(* PLC project project, Beckhoff Automation GmbH TwinCAT PLC Control 3.5.6.1 *)
(* stored: creationDateTime 2016-08-11T14:04:35.7870087, modificationDateTime 2016-08-11T14:04:35.7940091 *)

TYPE IOStruct :
STRUCT
	input_one : BOOL;
	input_two : BOOL;
	input_three : BOOL;
	input_four : BOOL;
	input_five : BOOL;
	input_six : BOOL;
END_STRUCT
END_TYPE

FUNCTION IO_aggregation : BOOL
VAR_INPUT
END_VAR
VAR
END_VAR

                  //Jedem Wert einen sensor zuweißen 
//Byte von 0-7; Position 0 am ende!!!!
//Z.B:

//IO_data.input_v.1 := GVL.in_MagazinNotaus;
//IO_data.input_one := NOT GVL.in_SortierbandNotaus;
//IO_data.input_two := NOT GVL.in_MagazinNotaus;
//IO_data.input_three := NOT GVL.in_StempelNotaus;
//IO_data.input_four := Main.Crane.Crane_SoftwareEmergency;
//IO_data.input_five := Main.Stamp.Stamp_SoftwareEmergency;
//IO_data.input_six := Main.PicAlpha.PicAlpha_SoftwareEmergency;
                
END_FUNCTION

PROGRAM MAIN
VAR		
	XPPU : XPPU;
END_VAR

                  XPPU();


//Für ADS
IO_aggregation();
                
END_PROGRAM

FUNCTION_BLOCK BistableCylinder
VAR_INPUT		
	SFCReset : BOOL;
END_VAR
VAR_OUTPUT
END_VAR
VAR	
	DI_Extended AT %I* : BOOL;
	DI_Retracted AT %I* : BOOL;
	DO_Extend AT %Q* : BOOL;
	DO_Retract AT %Q* : BOOL;
END_VAR

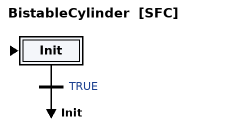
INITIAL_STEP Init:
END_STEP
TRANSITION FROM Init TO Init
  := TRUE;
END_TRANSITION

ACTION ACT_Retract:
                      DO_Extend:=FALSE;
DO_Retract:=TRUE;
                    
END_ACTION

ACTION ACT_Extend:
                      DO_Retract:=FALSE;
DO_Extend:=TRUE;
                    
END_ACTION
END_FUNCTION_BLOCK

FUNCTION_BLOCK MonostableCylinder
VAR_INPUT	
	SFCReset : BOOL;
END_VAR	
VAR_OUTPUT	
END_VAR
VAR	
	DI_Extended AT %I* : BOOL;
	DI_Retracted AT %I* : BOOL;
	
	DO_Extend AT %Q* : BOOL;
END_VAR

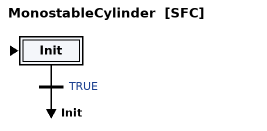
INITIAL_STEP Init:
END_STEP
TRANSITION FROM Init TO Init
  := TRUE;
END_TRANSITION

ACTION ACT_Extend:
                      DO_Extend:=TRUE;
                    
END_ACTION

ACTION ACT_Retract:
                      DO_Extend:=FALSE;
                    
END_ACTION
END_FUNCTION_BLOCK

FUNCTION_BLOCK Motor
VAR_INPUT	
	SFCReset : BOOL;
END_VAR
VAR_OUTPUT	
END_VAR
VAR	
	//Hardware
	DO_Forwards AT %Q* : BOOL;
	DO_Backwards AT %Q* : BOOL;
END_VAR

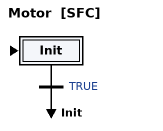
INITIAL_STEP Init:
END_STEP
TRANSITION FROM Init TO Init
  := TRUE;
END_TRANSITION

ACTION ACT_TurnBackwards:
                      DO_Forwards:=FALSE;
DO_Backwards:=TRUE;
                    
END_ACTION

ACTION ACT_Stop:
                      DO_Forwards:=FALSE;
DO_Backwards:=FALSE;
                    
END_ACTION

ACTION ACT_TurnForwards:
                      DO_Backwards:=FALSE;
DO_Forwards:=TRUE;
                    
END_ACTION
END_FUNCTION_BLOCK

FUNCTION_BLOCK Switch
VAR_INPUT	
	SFCReset : BOOL;
END_VAR	
VAR_OUTPUT		
END_VAR
VAR	
	//Hardware
	DI_Extended AT %I* : BOOL;
	DI_Retracted AT %I* : BOOL;	
	DO_Extend AT %Q* : BOOL;
END_VAR

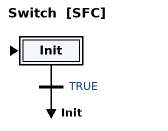
INITIAL_STEP Init:
END_STEP
TRANSITION FROM Init TO Init
  := TRUE;
END_TRANSITION

ACTION ACT_Extend:
                      DO_Extend:=TRUE;
                    
END_ACTION

ACTION ACT_Retract:
                      DO_Extend:=FALSE;
                    
END_ACTION
END_FUNCTION_BLOCK

FUNCTION_BLOCK VacuumGripper
VAR_INPUT	
	SFCReset : BOOL;
END_VAR
VAR_OUTPUT	
END_VAR
VAR	
	//Hardware
	DI_TakenIn AT %I* : BOOL;
	DO_Intake AT %Q* : BOOL;
END_VAR

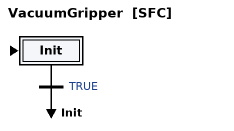
INITIAL_STEP Init:
END_STEP
TRANSITION FROM Init TO Init
  := TRUE;
END_TRANSITION

ACTION ACT_Intake:
                      DO_Intake:=TRUE;
                    
END_ACTION

ACTION ACT_Release:
                      DO_Intake:=FALSE;
                    
END_ACTION
END_FUNCTION_BLOCK

FUNCTION_BLOCK Crane
VAR_INPUT
	LiftingCylinder : MonostableCylinder;
	Gripper : VacuumGripper;			
	//Software
	Crane_SoftwareEmergency : BOOL;
	SFCReset : BOOL;
	InitCompleted : BOOL;
	LSC_AllowedToOperate : BOOL;
	Stamp_AllowedToOperate : BOOL;
	EmergencyHandeled : BOOL;	
END_VAR
VAR_OUTPUT	
	//Software
	Crane_WPPickedUp : BOOL;
	Crane_WPWeight_Light : BOOL;
	Crane_WPWeight_Medium : BOOL;
	Crane_WPWeight_Heavy : BOOL;
	AtStack : BOOL := FALSE;
	AtConveyor : BOOL := FALSE;
	AtStamp : BOOL := FALSE;	
END_VAR
VAR		
	//Hardware	
	Crane_OnStack AT %I* : BOOL;
	Crane_OnConveyor AT %I* : BOOL;
	Crane_OnStamp AT %I* : BOOL;	
	CraneTurnClockwise AT %Q* : BOOL;
	CraneTurnCounterclockwise AT %Q* : BOOL;
	
	//Software
	Timer : TON;	
	AutomaticExecuteAktive : BOOL;
END_VAR

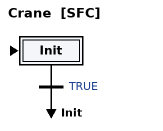
INITIAL_STEP Init:
END_STEP
TRANSITION FROM Init TO Init
  := TRUE;
END_TRANSITION

ACTION ACT_EmergencyStop:
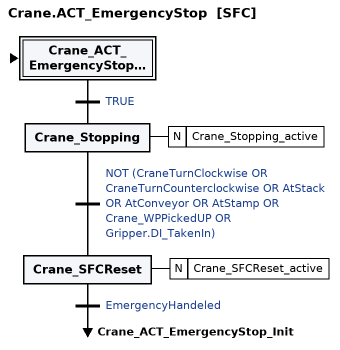
INITIAL_STEP Crane_ACT_EmergencyStop_Init:
END_STEP
TRANSITION FROM Crane_ACT_EmergencyStop_Init TO Crane_Stopping
  := TRUE;
END_TRANSITION
STEP Crane_Stopping:
  Crane_Stopping_active(N);
END_STEP
TRANSITION FROM Crane_Stopping TO Crane_SFCReset
  := NOT (CraneTurnClockwise OR CraneTurnCounterclockwise OR AtStack OR AtConveyor OR AtStamp OR Crane_WPPickedUP OR Gripper.DI_TakenIn);
END_TRANSITION
STEP Crane_SFCReset:
  Crane_SFCReset_active(N);
END_STEP
TRANSITION FROM Crane_SFCReset TO Crane_ACT_EmergencyStop_Init
  := EmergencyHandeled;
END_TRANSITION
END_ACTION

ACTION ACT_AutomaticExecute:
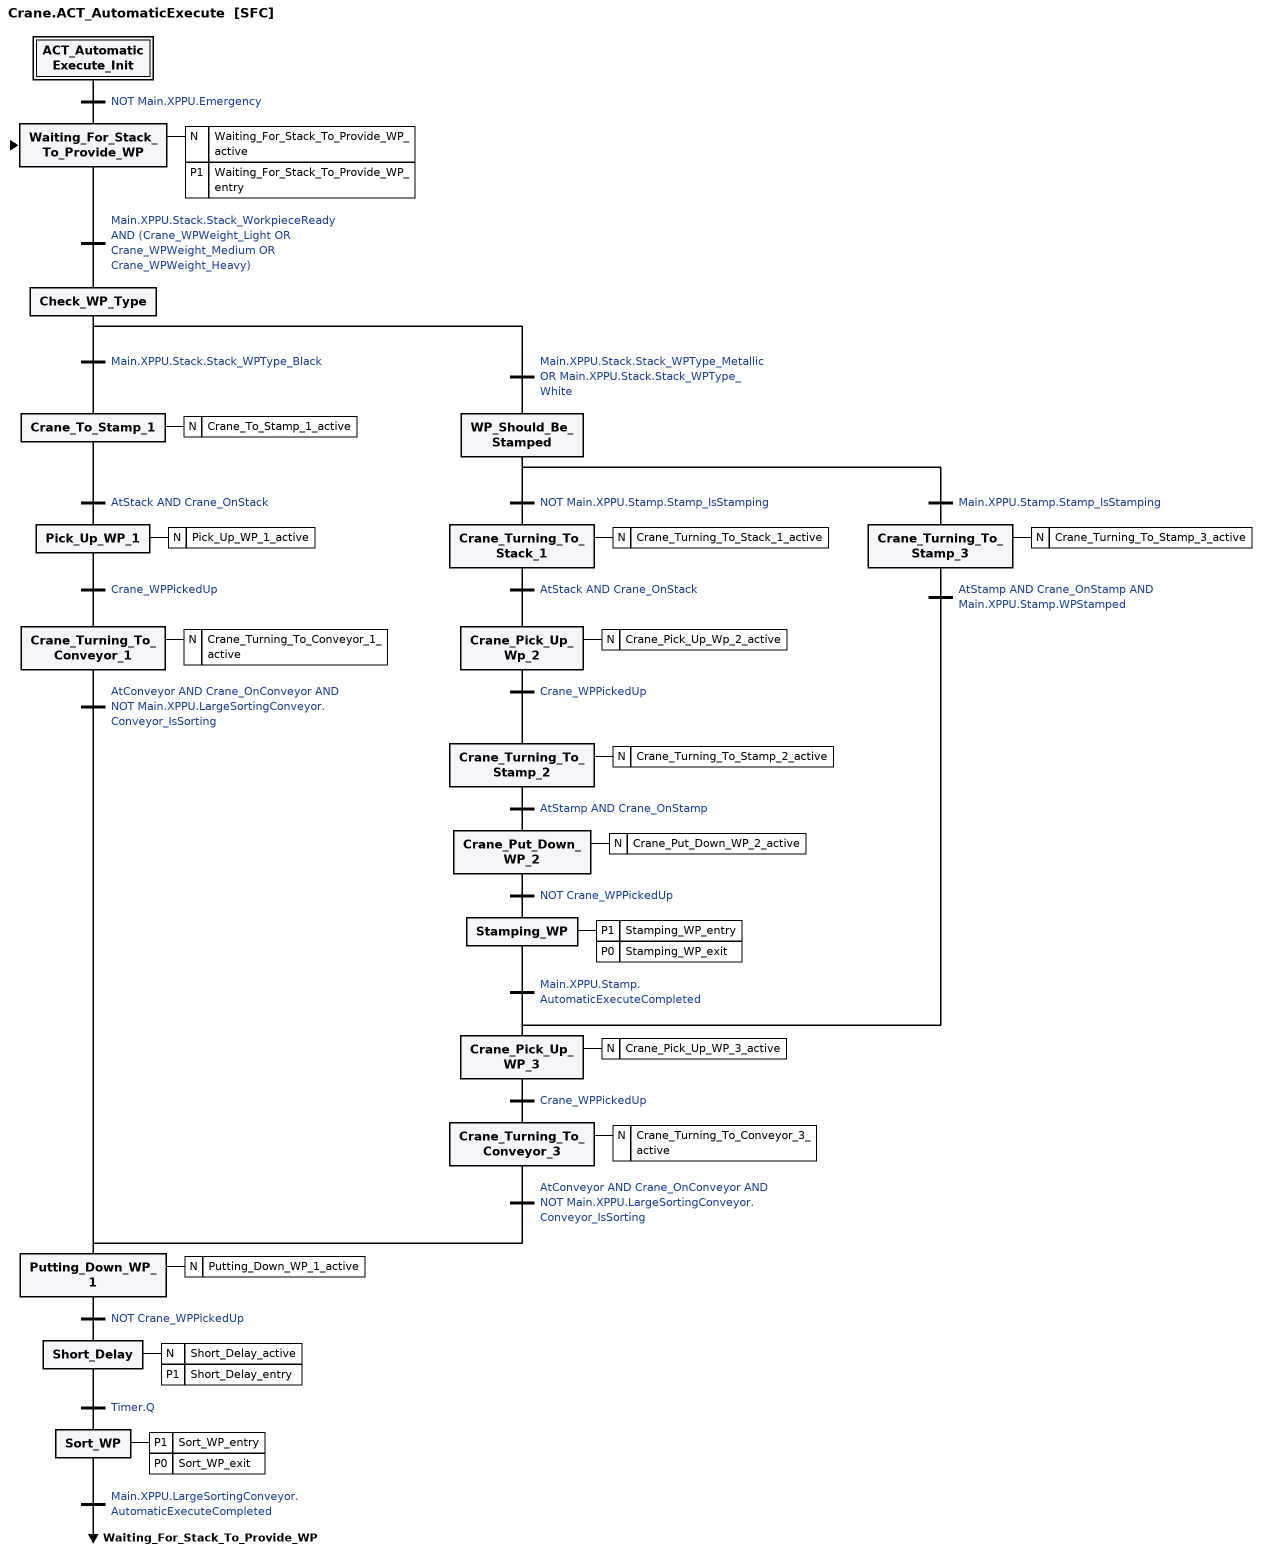
INITIAL_STEP ACT_AutomaticExecute_Init:
END_STEP
TRANSITION FROM ACT_AutomaticExecute_Init TO Waiting_For_Stack_To_Provide_WP
  := NOT Main.XPPU.Emergency;
END_TRANSITION
STEP Waiting_For_Stack_To_Provide_WP:
  Waiting_For_Stack_To_Provide_WP_active(N);
  Waiting_For_Stack_To_Provide_WP_entry(P1);
END_STEP
TRANSITION FROM Waiting_For_Stack_To_Provide_WP TO Check_WP_Type
  := Main.XPPU.Stack.Stack_WorkpieceReady AND (Crane_WPWeight_Light OR Crane_WPWeight_Medium OR Crane_WPWeight_Heavy);
END_TRANSITION
STEP Check_WP_Type:
END_STEP
TRANSITION FROM Check_WP_Type TO Crane_To_Stamp_1
  := Main.XPPU.Stack.Stack_WPType_Black;
END_TRANSITION
TRANSITION FROM Check_WP_Type TO WP_Should_Be_Stamped
  := Main.XPPU.Stack.Stack_WPType_Metallic OR Main.XPPU.Stack.Stack_WPType_White;
END_TRANSITION
STEP Crane_To_Stamp_1:
  Crane_To_Stamp_1_active(N);
END_STEP
TRANSITION FROM Crane_To_Stamp_1 TO Pick_Up_WP_1
  := AtStack AND Crane_OnStack;
END_TRANSITION
STEP Pick_Up_WP_1:
  Pick_Up_WP_1_active(N);
END_STEP
TRANSITION FROM Pick_Up_WP_1 TO Crane_Turning_To_Conveyor_1
  := Crane_WPPickedUp;
END_TRANSITION
STEP Crane_Turning_To_Conveyor_1:
  Crane_Turning_To_Conveyor_1_active(N);
END_STEP
TRANSITION FROM Crane_Turning_To_Conveyor_1 TO Putting_Down_WP_1
  := AtConveyor AND Crane_OnConveyor AND NOT Main.XPPU.LargeSortingConveyor.Conveyor_IsSorting;
END_TRANSITION
STEP Putting_Down_WP_1:
  Putting_Down_WP_1_active(N);
END_STEP
TRANSITION FROM Putting_Down_WP_1 TO Short_Delay
  := NOT Crane_WPPickedUp;
END_TRANSITION
STEP Short_Delay:
  Short_Delay_active(N);
  Short_Delay_entry(P1);
END_STEP
TRANSITION FROM Short_Delay TO Sort_WP
  := Timer.Q;
END_TRANSITION
STEP Sort_WP:
  Sort_WP_entry(P1);
  Sort_WP_exit(P0);
END_STEP
TRANSITION FROM Sort_WP TO Waiting_For_Stack_To_Provide_WP
  := Main.XPPU.LargeSortingConveyor.AutomaticExecuteCompleted;
END_TRANSITION
STEP WP_Should_Be_Stamped:
END_STEP
TRANSITION FROM WP_Should_Be_Stamped TO Crane_Turning_To_Stack_1
  := NOT Main.XPPU.Stamp.Stamp_IsStamping;
END_TRANSITION
TRANSITION FROM WP_Should_Be_Stamped TO Crane_Turning_To_Stamp_3
  := Main.XPPU.Stamp.Stamp_IsStamping;
END_TRANSITION
STEP Crane_Turning_To_Stack_1:
  Crane_Turning_To_Stack_1_active(N);
END_STEP
TRANSITION FROM Crane_Turning_To_Stack_1 TO Crane_Pick_Up_Wp_2
  := AtStack AND Crane_OnStack;
END_TRANSITION
STEP Crane_Pick_Up_Wp_2:
  Crane_Pick_Up_Wp_2_active(N);
END_STEP
TRANSITION FROM Crane_Pick_Up_Wp_2 TO Crane_Turning_To_Stamp_2
  := Crane_WPPickedUp;
END_TRANSITION
STEP Crane_Turning_To_Stamp_2:
  Crane_Turning_To_Stamp_2_active(N);
END_STEP
TRANSITION FROM Crane_Turning_To_Stamp_2 TO Crane_Put_Down_WP_2
  := AtStamp AND Crane_OnStamp;
END_TRANSITION
STEP Crane_Put_Down_WP_2:
  Crane_Put_Down_WP_2_active(N);
END_STEP
TRANSITION FROM Crane_Put_Down_WP_2 TO Stamping_WP
  := NOT Crane_WPPickedUp;
END_TRANSITION
STEP Stamping_WP:
  Stamping_WP_entry(P1);
  Stamping_WP_exit(P0);
END_STEP
TRANSITION FROM Stamping_WP TO Crane_Pick_Up_WP_3
  := Main.XPPU.Stamp.AutomaticExecuteCompleted;
END_TRANSITION
STEP Crane_Turning_To_Stamp_3:
  Crane_Turning_To_Stamp_3_active(N);
END_STEP
TRANSITION FROM Crane_Turning_To_Stamp_3 TO Crane_Pick_Up_WP_3
  := AtStamp AND Crane_OnStamp AND Main.XPPU.Stamp.WPStamped;
END_TRANSITION
STEP Crane_Pick_Up_WP_3:
  Crane_Pick_Up_WP_3_active(N);
END_STEP
TRANSITION FROM Crane_Pick_Up_WP_3 TO Crane_Turning_To_Conveyor_3
  := Crane_WPPickedUp;
END_TRANSITION
STEP Crane_Turning_To_Conveyor_3:
  Crane_Turning_To_Conveyor_3_active(N);
END_STEP
TRANSITION FROM Crane_Turning_To_Conveyor_3 TO Putting_Down_WP_1
  := AtConveyor AND Crane_OnConveyor AND NOT Main.XPPU.LargeSortingConveyor.Conveyor_IsSorting;
END_TRANSITION
END_ACTION

ACTION ACT_Init:
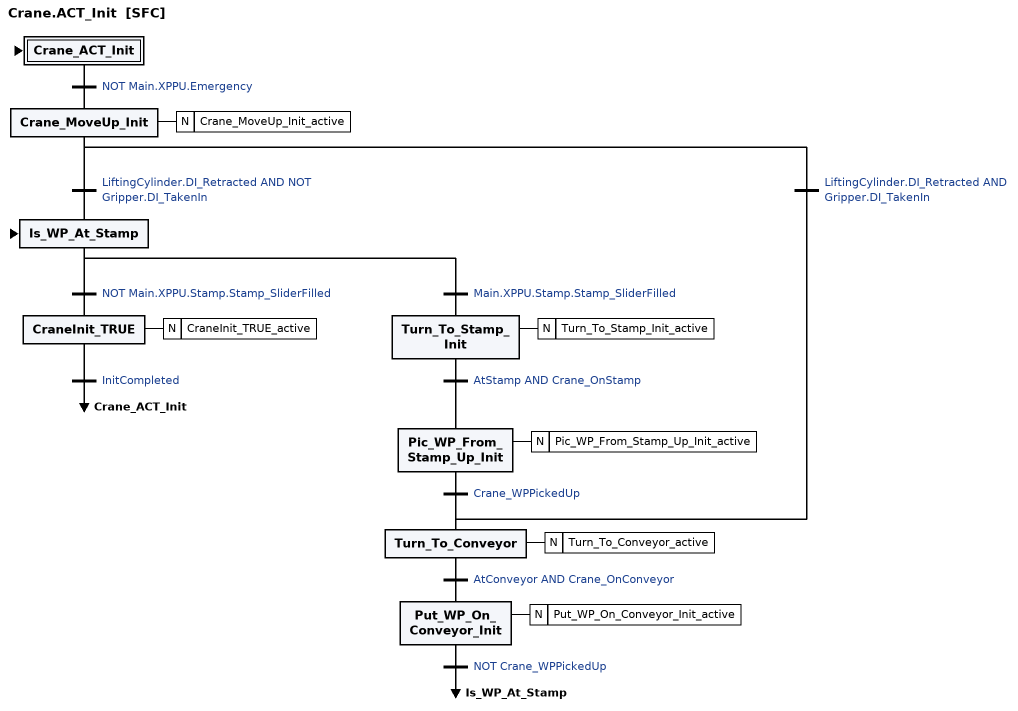
INITIAL_STEP Crane_ACT_Init:
END_STEP
TRANSITION FROM Crane_ACT_Init TO Crane_MoveUp_Init
  := NOT Main.XPPU.Emergency;
END_TRANSITION
STEP Crane_MoveUp_Init:
  Crane_MoveUp_Init_active(N);
END_STEP
TRANSITION FROM Crane_MoveUp_Init TO Is_WP_At_Stamp
  := LiftingCylinder.DI_Retracted AND NOT Gripper.DI_TakenIn;
END_TRANSITION
TRANSITION FROM Crane_MoveUp_Init TO Turn_To_Conveyor
  := LiftingCylinder.DI_Retracted AND Gripper.DI_TakenIn;
END_TRANSITION
STEP Turn_To_Conveyor:
  Turn_To_Conveyor_active(N);
END_STEP
TRANSITION FROM Turn_To_Conveyor TO Put_WP_On_Conveyor_Init
  := AtConveyor AND Crane_OnConveyor;
END_TRANSITION
STEP Put_WP_On_Conveyor_Init:
  Put_WP_On_Conveyor_Init_active(N);
END_STEP
TRANSITION FROM Put_WP_On_Conveyor_Init TO Is_WP_At_Stamp
  := NOT Crane_WPPickedUp;
END_TRANSITION
STEP Is_WP_At_Stamp:
END_STEP
TRANSITION FROM Is_WP_At_Stamp TO CraneInit_TRUE
  := NOT Main.XPPU.Stamp.Stamp_SliderFilled;
END_TRANSITION
TRANSITION FROM Is_WP_At_Stamp TO Turn_To_Stamp_Init
  := Main.XPPU.Stamp.Stamp_SliderFilled;
END_TRANSITION
STEP Turn_To_Stamp_Init:
  Turn_To_Stamp_Init_active(N);
END_STEP
TRANSITION FROM Turn_To_Stamp_Init TO Pic_WP_From_Stamp_Up_Init
  := AtStamp AND Crane_OnStamp;
END_TRANSITION
STEP Pic_WP_From_Stamp_Up_Init:
  Pic_WP_From_Stamp_Up_Init_active(N);
END_STEP
TRANSITION FROM Pic_WP_From_Stamp_Up_Init TO Turn_To_Conveyor
  := Crane_WPPickedUp;
END_TRANSITION
STEP CraneInit_TRUE:
  CraneInit_TRUE_active(N);
END_STEP
TRANSITION FROM CraneInit_TRUE TO Crane_ACT_Init
  := InitCompleted;
END_TRANSITION
END_ACTION

ACTION Delay_Heavy_active:
                      Timer(IN:=TRUE, PT:=T#2000ms);
                    
END_ACTION

ACTION Sort_WP_1_exit:
                      LSC_AllowedToOperate:=FALSE;
                    
END_ACTION

ACTION Turn_To_Stamp_Init_active:
                      ACT_MoveToStamp();
                    
END_ACTION

ACTION Delay_Light_entry:
                      Timer(IN:=FALSE);
                    
END_ACTION

ACTION Set_Value_active:
                      Crane_WPPickedUp:=TRUE;
                    
END_ACTION

ACTION Crane_SFCReset_active:
                      EmergencyHandeled:=TRUE;	


                    
END_ACTION

ACTION Crane_Pick_Up_WP_3_active:
                      ACT_PickUpWP();
                    
END_ACTION

ACTION Set_Value_active_0:
                      Crane_WPPickedUp:=FALSE;
                    
END_ACTION

ACTION Turn_On_Vacuum_PWU_entry:
                      Timer(IN:=FALSE);
                    
END_ACTION

ACTION Crane_MoveUp_Init_active:
                      LiftingCylinder.ACT_Retract();
                    
END_ACTION

ACTION Crane_Turning_To_Conveyor_1_active:
                      ACT_MoveToConveyor();
                    
END_ACTION

ACTION Delay_Medium_entry:
                      Timer(IN:=FALSE);
                    
END_ACTION

ACTION Error_active:
                      LiftingCylinder.ACT_Retract();
Crane_SoftwareEmergency:=true;
                    
END_ACTION

ACTION AutomaticExecute_active:
                      ACT_AutomaticExecute();
                    
END_ACTION

ACTION Sort_WP_1_entry:
                      LSC_AllowedToOperate:=TRUE;
                    
END_ACTION

ACTION DecideHowToMoveCrane_entry:
                      AtConveyor:=FALSE;
                    
END_ACTION

ACTION Crane_Turning_To_Stamp_3_active:
                      ACT_MoveToStamp();
                    
END_ACTION

ACTION CraneStop_MTS_exit:
                      AtStamp:=TRUE;
                    
END_ACTION

ACTION Crane_VacuumOff_Init_active:
                      Gripper.ACT_Release();
                    
END_ACTION

ACTION Turn_CounterClockwise_active_0:
                      CraneTurnClockwise:=FALSE;
CraneTurnCounterclockwise:=TRUE;
                    
END_ACTION

ACTION Move_Crane_Up_active_0:
                      LiftingCylinder.ACT_Retract();
                    
END_ACTION

ACTION Crane_To_Stamp_1_active:
                      ACT_MoveToStack();
                    
END_ACTION

ACTION Turn_Clockwise_MTM_entry:
                      ATStack:=FALSE;
                    
END_ACTION

ACTION Turn_CounterClockwise_MTS_entry:
                      AtStamp:=FALSE;
                    
END_ACTION

ACTION Crane_Pick_Up_Wp_2_active:
                      ACT_PickUpWP();
                    
END_ACTION

ACTION Sort_WP_exit:
                      LSC_AllowedToOperate:=False;
                    
END_ACTION

ACTION Crane_Put_Down_WP_2_active:
                      ACT_PutDownWP();
                    
END_ACTION

ACTION CraneStop_MTS_active:
                      CraneTurnClockwise:=FALSE;
CraneTurnCounterclockwise:=FALSE;
                    
END_ACTION

ACTION Short_Delay_active:
                      Timer(IN:=TRUE, PT:=T#50ms);
                    
END_ACTION

ACTION Stop_Crane_active:
                      CraneTurnClockwise:=FALSE;
CraneTurnCounterclockwise:=FALSE;
                    
END_ACTION

ACTION StopCrane_MTM_active:
                      CraneTurnClockwise:=FALSE;
CraneTurnCounterclockwise:=FALSE;
                    
END_ACTION

ACTION Lower_Crane_active:
                      LiftingCylinder.ACT_Extend();
                    
END_ACTION

ACTION Stamping_WP_exit:
                      Stamp_AllowedToOperate:=FALSE;
                    
END_ACTION

ACTION Crane_Stop_Init_active:
                      CraneTurnClockwise:=FALSE;
CraneTurnCounterclockwise:=FALSE;
                    
END_ACTION

ACTION Reset_Timer_active:
                      Timer(In:=FALSE);
                    
END_ACTION

ACTION Short_Delay_entry:
                      Timer(IN:=FALSE);
                    
END_ACTION

ACTION Crane_Turning_To_Stack_1_active:
                      ACT_MoveToStack();
                    
END_ACTION

ACTION Crane_Turning_To_Conveyor_3_active:
                      ACT_MoveToConveyor();
                    
END_ACTION

ACTION CraneInit_TRUE_active:
                      InitCompleted:=TRUE;
                    
END_ACTION

ACTION Waiting_For_Stack_To_Provide_WP_active:
                      IF(Main.XPPU.Stack.Stack_WPWeight_Light) THEN
	Crane_WPWeight_Light:=TRUE;
	Crane_WPWeight_Medium:=FALSE;
	Crane_WPWeight_Heavy:=FALSE;
ELSIF(Main.XPPU.Stack.Stack_WPWeight_Medium)THEN
	Crane_WPWeight_Light:=FALSE;
	Crane_WPWeight_Medium:=TRUE;
	Crane_WPWeight_Heavy:=FALSE;
ELSIF(Main.XPPU.Stack.Stack_WPWeight_Heavy)THEN
	Crane_WPWeight_Light:=FALSE;
	Crane_WPWeight_Medium:=FALSE;
	Crane_WPWeight_Heavy:=TRUE;
END_IF
                    
END_ACTION

ACTION Delay_Medium_active:
                      Timer(IN:=TRUE, PT:=T#1000ms);
                    
END_ACTION

ACTION EmergencyStop_active:
                      
ACT_EmergencyStop();

                    
END_ACTION

ACTION Delay_Light_active:
                      Timer(IN:=TRUE, PT:=T#0ms);
                    
END_ACTION

ACTION First_Turn_CounterC_entry:
                      Timer(IN:=FALSE);
                    
END_ACTION

ACTION Waiting_For_Stack_To_Provide_WP_entry:
                      Crane_WPWeight_Light:=FALSE;
Crane_WPWeight_Medium:=FALSE;
Crane_WPWeight_Heavy:=FALSE;
                    
END_ACTION

ACTION Second_Turn_Clockwise_active:
                      CraneTurnCounterClockwise:=FALSE;
CraneTurnClockwise:=TRUE;


                    
END_ACTION

ACTION Turn_To_Conveyor_active:
                      Crane_WPPickedUp:=TRUE;
ACT_MoveToConveyor();
                    
END_ACTION

ACTION Stamping_WP_entry:
                      Stamp_AllowedToOperate:=TRUE;
                    
END_ACTION

ACTION Putting_Down_WP_1_active:
                      ACT_PutDownWP();
                    
END_ACTION

ACTION Stamping_WP_active:
                      MAIN.XPPU.Stamp.ACT_Stamp();
                    
END_ACTION

ACTION First_Turn_CounterC_active:
                      CraneTurnClockwise:=FALSE;
CraneTurnCounterClockwise:=TRUE;
Timer(IN:=TRUE, PT:= T#5S);

                    
END_ACTION

ACTION Crane_Turning_To_Stamp_2_active:
                      ACT_MoveToStamp();
                    
END_ACTION

ACTION Turn_On_Vacuum_active:
                      Gripper.ACT_Intake();	
Timer(IN:=TRUE, PT:=T#2s);
                    
END_ACTION

ACTION Sort_WP_entry:
                      LSC_AllowedToOperate:=TRUE;
                    
END_ACTION

ACTION Lower_Crane_active_0:
                      LiftingCylinder.ACT_Extend();
                    
END_ACTION

ACTION Turn_CLockwise_active:
                      CraneTurnCounterclockwise:=FALSE;
CraneTurnClockwise:=TRUE;
                    
END_ACTION

ACTION Crane_Stopping_active:
                      Crane_WPPickedUp:=FALSE;
AtStack:=FALSE;
AtConveyor:=FALSE;
AtStamp:=FALSE;

CraneTurnClockwise:=FALSE;
CraneTurnCounterclockwise:=FALSE;
Gripper.ACT_Release();
                    
END_ACTION

ACTION Turn_Clockwise_active_0:
                      CraneTurnCounterclockwise:=FALSE;
CraneTurnClockwise:=TRUE;

                    
END_ACTION

ACTION CraneInit_FALSE_active:
                      InitCompleted:=FALSE;
                    
END_ACTION

ACTION Put_WP_On_Conveyor_Init_active:
                      ACT_PutDownWP();
                    
END_ACTION

ACTION Move_Crane_Up_active:
                      LiftingCylinder.ACT_Retract();
                    
END_ACTION

ACTION Delay_Heavy_entry:
                      Timer(IN:=FALSE);
                    
END_ACTION

ACTION StopCrane_MTC_exit:
                      ATConveyor:=TRUE;
                    
END_ACTION

ACTION StopCrane_MTM_exit:
                      AtStack:=TRUE;
                    
END_ACTION

ACTION Pic_WP_From_Stamp_Up_Init_active:
                      ACT_PickUpWP();
                    
END_ACTION

ACTION Pick_Up_WP_1_active:
                      ACT_PickUpWP();
                    
END_ACTION

ACTION Turn_CounterClockwise_active:
                      CraneTurnClockwise:=FALSE;
CraneTurnCounterclockwise:=TRUE;
                    
END_ACTION

ACTION Put_WP_Down_active:
                      Gripper.ACT_Release();
                    
END_ACTION

ACTION ACT_PickUpWP:
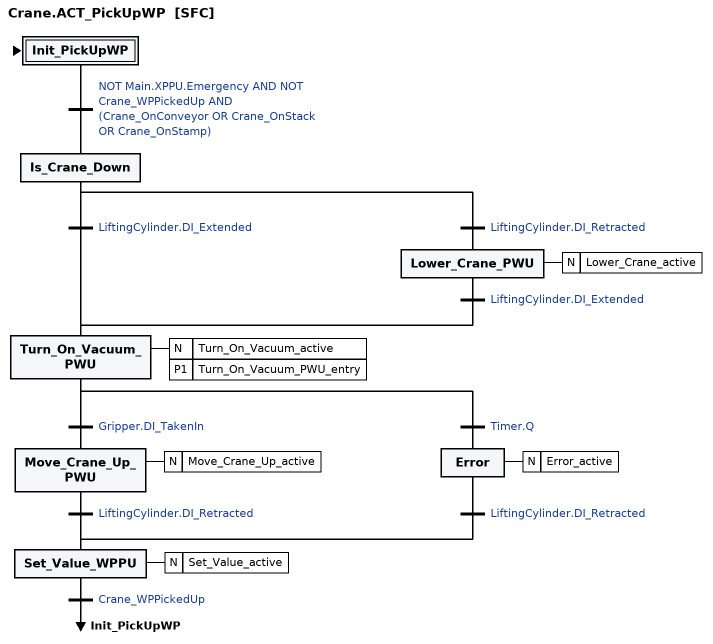
INITIAL_STEP Init_PickUpWP:
END_STEP
TRANSITION FROM Init_PickUpWP TO Is_Crane_Down
  := NOT Main.XPPU.Emergency AND NOT Crane_WPPickedUp AND (Crane_OnConveyor OR Crane_OnStack OR Crane_OnStamp);
END_TRANSITION
STEP Is_Crane_Down:
END_STEP
TRANSITION FROM Is_Crane_Down TO Turn_On_Vacuum_PWU
  := LiftingCylinder.DI_Extended;
END_TRANSITION
TRANSITION FROM Is_Crane_Down TO Lower_Crane_PWU
  := LiftingCylinder.DI_Retracted;
END_TRANSITION
STEP Lower_Crane_PWU:
  Lower_Crane_active(N);
END_STEP
TRANSITION FROM Lower_Crane_PWU TO Turn_On_Vacuum_PWU
  := LiftingCylinder.DI_Extended;
END_TRANSITION
STEP Turn_On_Vacuum_PWU:
  Turn_On_Vacuum_active(N);
  Turn_On_Vacuum_PWU_entry(P1);
END_STEP
TRANSITION FROM Turn_On_Vacuum_PWU TO Move_Crane_Up_PWU
  := Gripper.DI_TakenIn;
END_TRANSITION
TRANSITION FROM Turn_On_Vacuum_PWU TO Error
  := Timer.Q;
END_TRANSITION
STEP Move_Crane_Up_PWU:
  Move_Crane_Up_active(N);
END_STEP
TRANSITION FROM Move_Crane_Up_PWU TO Set_Value_WPPU
  := LiftingCylinder.DI_Retracted;
END_TRANSITION
STEP Error:
  Error_active(N);
END_STEP
TRANSITION FROM Error TO Set_Value_WPPU
  := LiftingCylinder.DI_Retracted;
END_TRANSITION
STEP Set_Value_WPPU:
  Set_Value_active(N);
END_STEP
TRANSITION FROM Set_Value_WPPU TO Init_PickUpWP
  := Crane_WPPickedUp;
END_TRANSITION
END_ACTION

ACTION ACT_PutDownWP:
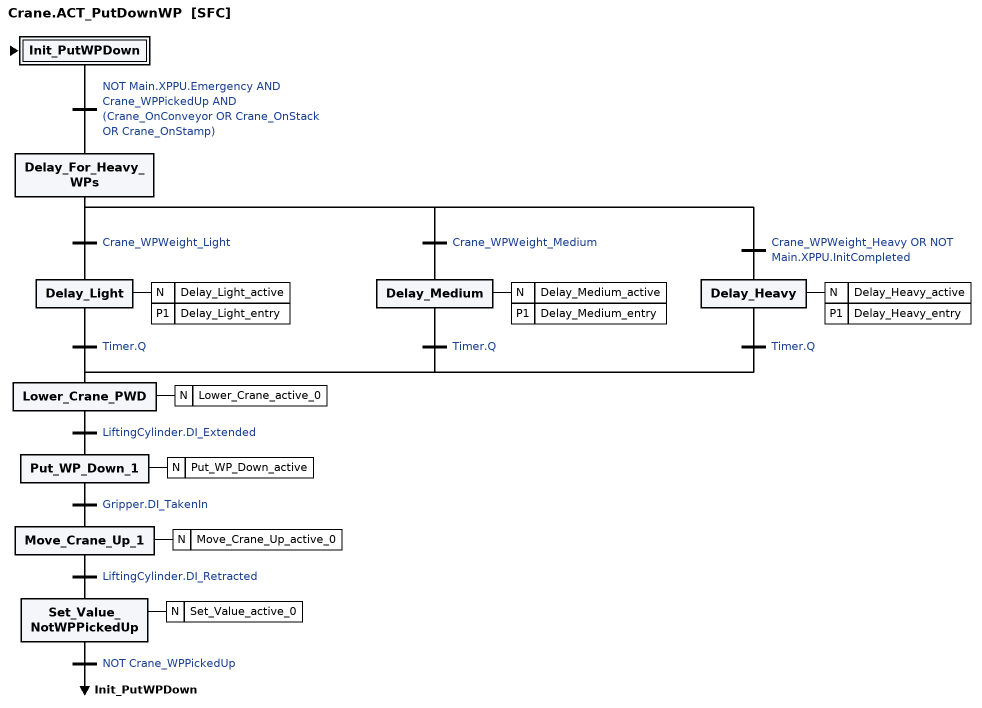
INITIAL_STEP Init_PutWPDown:
END_STEP
TRANSITION FROM Init_PutWPDown TO Delay_For_Heavy_WPs
  := NOT Main.XPPU.Emergency AND Crane_WPPickedUp AND (Crane_OnConveyor OR Crane_OnStack OR Crane_OnStamp);
END_TRANSITION
STEP Delay_For_Heavy_WPs:
END_STEP
TRANSITION FROM Delay_For_Heavy_WPs TO Delay_Light
  := Crane_WPWeight_Light;
END_TRANSITION
TRANSITION FROM Delay_For_Heavy_WPs TO Delay_Medium
  := Crane_WPWeight_Medium;
END_TRANSITION
TRANSITION FROM Delay_For_Heavy_WPs TO Delay_Heavy
  := Crane_WPWeight_Heavy OR NOT Main.XPPU.InitCompleted;
END_TRANSITION
STEP Delay_Light:
  Delay_Light_active(N);
  Delay_Light_entry(P1);
END_STEP
TRANSITION FROM Delay_Light TO Lower_Crane_PWD
  := Timer.Q;
END_TRANSITION
STEP Delay_Medium:
  Delay_Medium_active(N);
  Delay_Medium_entry(P1);
END_STEP
TRANSITION FROM Delay_Medium TO Lower_Crane_PWD
  := Timer.Q;
END_TRANSITION
STEP Delay_Heavy:
  Delay_Heavy_active(N);
  Delay_Heavy_entry(P1);
END_STEP
TRANSITION FROM Delay_Heavy TO Lower_Crane_PWD
  := Timer.Q;
END_TRANSITION
STEP Lower_Crane_PWD:
  Lower_Crane_active_0(N);
END_STEP
TRANSITION FROM Lower_Crane_PWD TO Put_WP_Down_1
  := LiftingCylinder.DI_Extended;
END_TRANSITION
STEP Put_WP_Down_1:
  Put_WP_Down_active(N);
END_STEP
TRANSITION FROM Put_WP_Down_1 TO Move_Crane_Up_1
  := Gripper.DI_TakenIn;
END_TRANSITION
STEP Move_Crane_Up_1:
  Move_Crane_Up_active_0(N);
END_STEP
TRANSITION FROM Move_Crane_Up_1 TO Set_Value_NotWPPickedUp
  := LiftingCylinder.DI_Retracted;
END_TRANSITION
STEP Set_Value_NotWPPickedUp:
  Set_Value_active_0(N);
END_STEP
TRANSITION FROM Set_Value_NotWPPickedUp TO Init_PutWPDown
  := NOT Crane_WPPickedUp;
END_TRANSITION
END_ACTION

ACTION ACT_MoveToConveyor:
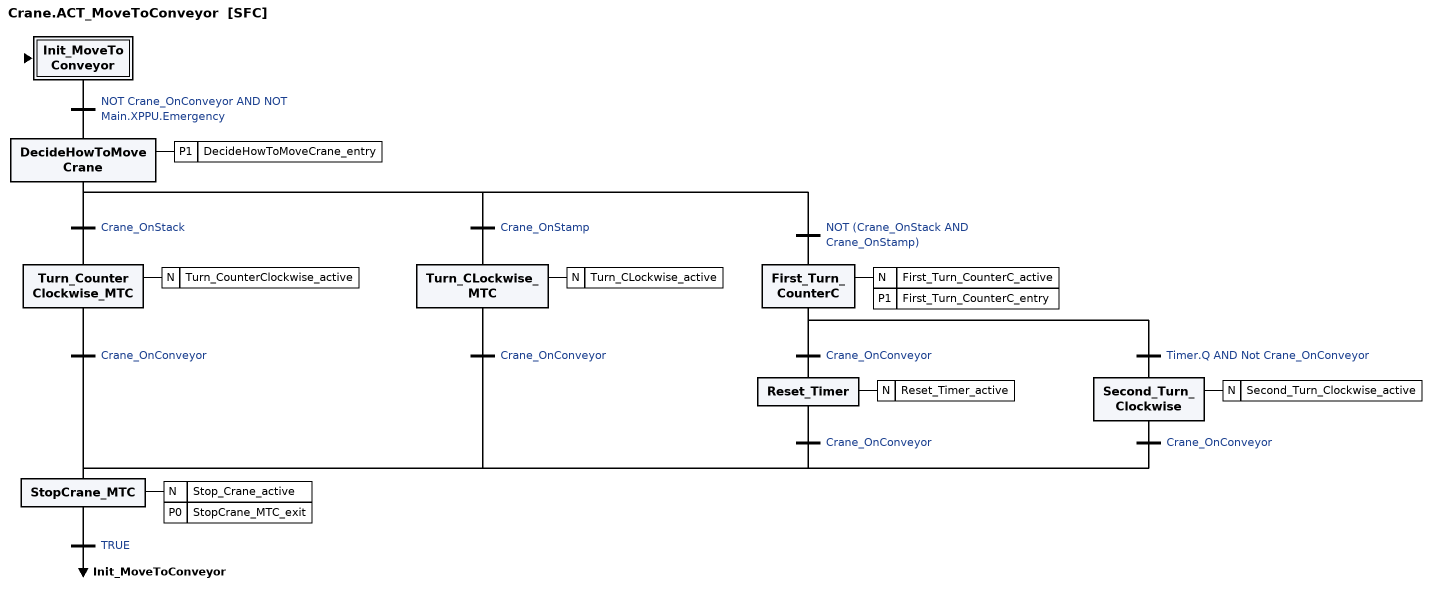
INITIAL_STEP Init_MoveToConveyor:
END_STEP
TRANSITION FROM Init_MoveToConveyor TO DecideHowToMoveCrane
  := NOT Crane_OnConveyor AND NOT Main.XPPU.Emergency;
END_TRANSITION
STEP DecideHowToMoveCrane:
  DecideHowToMoveCrane_entry(P1);
END_STEP
TRANSITION FROM DecideHowToMoveCrane TO Turn_CounterClockwise_MTC
  := Crane_OnStack;
END_TRANSITION
TRANSITION FROM DecideHowToMoveCrane TO Turn_CLockwise_MTC
  := Crane_OnStamp;
END_TRANSITION
TRANSITION FROM DecideHowToMoveCrane TO First_Turn_CounterC
  := NOT (Crane_OnStack AND Crane_OnStamp);
END_TRANSITION
STEP Turn_CounterClockwise_MTC:
  Turn_CounterClockwise_active(N);
END_STEP
TRANSITION FROM Turn_CounterClockwise_MTC TO StopCrane_MTC
  := Crane_OnConveyor;
END_TRANSITION
STEP Turn_CLockwise_MTC:
  Turn_CLockwise_active(N);
END_STEP
TRANSITION FROM Turn_CLockwise_MTC TO StopCrane_MTC
  := Crane_OnConveyor;
END_TRANSITION
STEP First_Turn_CounterC:
  First_Turn_CounterC_active(N);
  First_Turn_CounterC_entry(P1);
END_STEP
TRANSITION FROM First_Turn_CounterC TO Reset_Timer
  := Crane_OnConveyor;
END_TRANSITION
TRANSITION FROM First_Turn_CounterC TO Second_Turn_Clockwise
  := Timer.Q AND Not Crane_OnConveyor;
END_TRANSITION
STEP Reset_Timer:
  Reset_Timer_active(N);
END_STEP
TRANSITION FROM Reset_Timer TO StopCrane_MTC
  := Crane_OnConveyor;
END_TRANSITION
STEP Second_Turn_Clockwise:
  Second_Turn_Clockwise_active(N);
END_STEP
TRANSITION FROM Second_Turn_Clockwise TO StopCrane_MTC
  := Crane_OnConveyor;
END_TRANSITION
STEP StopCrane_MTC:
  Stop_Crane_active(N);
  StopCrane_MTC_exit(P0);
END_STEP
TRANSITION FROM StopCrane_MTC TO Init_MoveToConveyor
  := TRUE;
END_TRANSITION
END_ACTION

ACTION ACT_MoveToStamp:
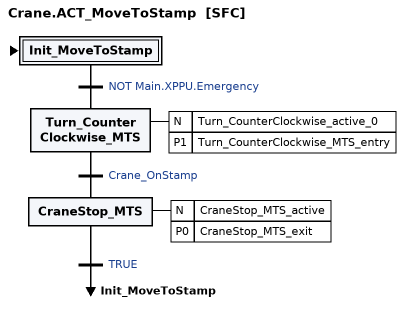
INITIAL_STEP Init_MoveToStamp:
END_STEP
TRANSITION FROM Init_MoveToStamp TO Turn_CounterClockwise_MTS
  := NOT Main.XPPU.Emergency;
END_TRANSITION
STEP Turn_CounterClockwise_MTS:
  Turn_CounterClockwise_active_0(N);
  Turn_CounterClockwise_MTS_entry(P1);
END_STEP
TRANSITION FROM Turn_CounterClockwise_MTS TO CraneStop_MTS
  := Crane_OnStamp;
END_TRANSITION
STEP CraneStop_MTS:
  CraneStop_MTS_active(N);
  CraneStop_MTS_exit(P0);
END_STEP
TRANSITION FROM CraneStop_MTS TO Init_MoveToStamp
  := TRUE;
END_TRANSITION
END_ACTION

ACTION ACT_MoveToStack:
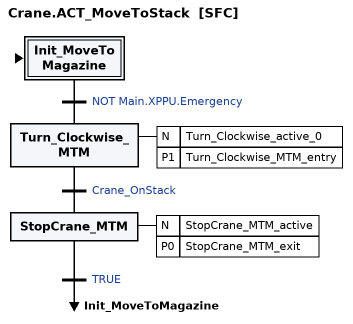
INITIAL_STEP Init_MoveToMagazine:
END_STEP
TRANSITION FROM Init_MoveToMagazine TO Turn_Clockwise_MTM
  := NOT Main.XPPU.Emergency;
END_TRANSITION
STEP Turn_Clockwise_MTM:
  Turn_Clockwise_active_0(N);
  Turn_Clockwise_MTM_entry(P1);
END_STEP
TRANSITION FROM Turn_Clockwise_MTM TO StopCrane_MTM
  := Crane_OnStack;
END_TRANSITION
STEP StopCrane_MTM:
  StopCrane_MTM_active(N);
  StopCrane_MTM_exit(P0);
END_STEP
TRANSITION FROM StopCrane_MTM TO Init_MoveToMagazine
  := TRUE;
END_TRANSITION
END_ACTION
END_FUNCTION_BLOCK

FUNCTION_BLOCK LargeSortingConveyor
VAR_INPUT
	Motor : Motor;
	Seperator1 : MonostableCylinder;
	Seperator2 : MonostableCylinder;
	//Software
	SFCReset : BOOL;
	InitCompleted : BOOL;
	AutomaticExecuteCompleted : BOOL;
	EmergencyHandeled : BOOL;	
END_VAR
VAR_OUTPUT			
	//Software	
	Conveyor_IsSorting : BOOL;
	Conveyor_WPSorted : BOOL;
	Conveyor_WPTypeChecked : BOOL;
	Conveyor_TargetChanged : BOOL;	
END_VAR
VAR	
	//Hardware	
	Conveyor_StartButton AT %I* : BOOL;
	Conveyor_EmergencyStop AT %I* : BOOL;		
	Conveyor_Beginning_PresenceSensor AT %I* : BOOL;
	Conveyor_Pusher1_InductiveSenor AT %I* : BOOL;
	Conveyor_Pusher1_OpticalSensor AT %I* : BOOL;	
	Conveyor_Ramp1_PresenceSensor AT %I* : BOOL;
	Conveyor_Pusher2_InductiveSenor AT %I* : BOOL;
	Conveyor_Pusher2_OpticalSensor AT %I* : BOOL;	
	Conveyor_Ramp2_PresenceSensor AT %I* : BOOL;
	Conveyor_Ramp3_OpticalSensor AT %I* : BOOL;
	Conveyor_Ramp3_PresenceSensor AT %I* : BOOL;
	ConveyorGreenLamp AT %Q* : BOOL;
	ConveyorWhiteLamp AT %Q* : BOOL;
	
	//Software
	Conveyor_WPType_White : BOOL;
	Conveyor_WPType_Black : BOOL;
	Conveyor_WPType_Metallic : BOOL;
	Conveyor_CurrentTarget_Ramp1 : BOOL;
	Conveyor_CurrentTarget_Ramp2 : BOOL;
	Conveyor_CurrentTarget_Ramp3 : BOOL;	
	Timer : TON;
END_VAR

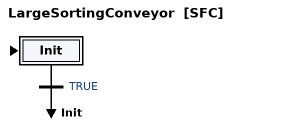
INITIAL_STEP Init:
END_STEP
TRANSITION FROM Init TO Init
  := TRUE;
END_TRANSITION

ACTION Conveyor_AutomaticExecute_Init_entry:
                      ConveyorWhiteLamp:=FALSE;
ConveyorGreenLamp:=TRUE;
                    
END_ACTION

ACTION Pusher2_Retract_active:
                      Seperator2.ACT_Retract();
                    
END_ACTION

ACTION ShortDelay_entry:
                      Timer(IN:=FALSE);
                    
END_ACTION

ACTION WP_Is_Sorted_active:
                      Conveyor_IsSorting:=FALSE;
Conveyor_WPSorted:=TRUE;
                    
END_ACTION

ACTION Conveyor_ACT_EmergencyStop_Init_entry:
                      ConveyorGreenLamp:=FALSE;
ConveyorWhiteLamp:=FALSE;
                    
END_ACTION

ACTION Stop_Conveyors_active:
                      Motor.ACT_Stop();
                    
END_ACTION

ACTION WP_Is_Metallic_active_0:
                      Conveyor_WPType_White:=FALSE;
Conveyor_WPType_Black:=FALSE;
Conveyor_WPType_Metallic:=TRUE;
                    
END_ACTION

ACTION Init_ACT_SortWP_entry:
                      
                    
END_ACTION

ACTION ConveyorPicAlpha_active:
                      
                    
END_ACTION

ACTION Transporting_To_Ramp1_entry:
                      Timer(IN:=FALSE);
                    
END_ACTION

ACTION WP_Type_Checked_active:
                      Conveyor_WPTypeChecked:=TRUE;
                    
END_ACTION

ACTION Start_Conveyor_PicAlpha_Init_active:
                      //Main.XPPU.ConveyorPicAlpha.ACT_MoveForwards();
Timer(IN:=TRUE, PT:=T#4s);
                    
END_ACTION

ACTION TurnConveyorOn_1_entry_0:
                      Timer(IN:=FALSE);
                    
END_ACTION

ACTION RampEnd_active_1:
                      Conveyor_CurrentTarget_Ramp3:=TRUE;
                    
END_ACTION

ACTION Pusher1_Retracting_active:
                      Seperator1.ACT_Retract();
                    
END_ACTION

ACTION Ramp1_active:
                      Conveyor_CurrentTarget_Ramp1:=TRUE;
                    
END_ACTION

ACTION ShortDelay_active_0:
                      Timer(IN:=TRUE, PT:=T#500ms);
                    
END_ACTION

ACTION Pusher1_Extending_active:
                      Seperator1.ACT_Extend();
                    
END_ACTION

ACTION RampEnd_active_0:
                      Conveyor_CurrentTarget_Ramp3:=TRUE;
                    
END_ACTION

ACTION RampEnd_active:
                      
                    
END_ACTION

ACTION Short_Delay_active:
                      Timer(IN:=FALSE, PT:=T#500ms);
                    
END_ACTION

ACTION Conveyor_To_Magazine_1_active:
                      Motor.ACT_TurnForwards();
                    
END_ACTION

ACTION WP_At_Beginning_entry:
                      Timer(IN:=FALSE);
                    
END_ACTION

ACTION TurnConveyorOn_1_exit:
                      Conveyor_WPType_White:=FALSE;
Conveyor_WPType_Black:=FALSE;
Conveyor_WPType_Metallic:=FALSE;

                    
END_ACTION

ACTION WP_At_Beginning_active:
                      
                    
END_ACTION

ACTION Conveyor_To_Magazine_1_entry:
                      Timer(IN:=FALSE);
                    
END_ACTION

ACTION WP_Is_Black_active:
                      Conveyor_WPType_White:=FALSE;
Conveyor_WPType_Black:=TRUE;
Conveyor_WPType_Metallic:=FALSE;
                    
END_ACTION

ACTION Conveyor_Sorting_active:
                      ACT_SortWP();
                    
END_ACTION

ACTION Pusher2_Extend_active:
                      Seperator2.ACT_Extend();
                    
END_ACTION

ACTION Ramp2_active:
                      
                    
END_ACTION

ACTION TurnConveyorOn_1_active:
                      Conveyor_WPSorted:=FALSE;
Conveyor_IsSorting:=TRUE;

Motor.ACT_TurnForwards();

Timer(IN:=TRUE, PT:=T#800ms);
                    
END_ACTION

ACTION Conveyor_ACT_CheckWPType_Init_exit:
                      Conveyor_WPTypeChecked:=FALSE;
                    
END_ACTION

ACTION Pusher1_Retracting_active_0:
                      Seperator1.ACT_Retract();
                    
END_ACTION

ACTION Conveyor_ACT_CheckWPType_Init_entry:
                      
                    
END_ACTION

ACTION WP_Is_White_active:
                      Conveyor_WPType_White:=TRUE;
Conveyor_WPType_Black:=FALSE;
Conveyor_WPType_Metallic:=FALSE;

                    
END_ACTION

ACTION Transporting_To_Ramp2_entry:
                      Timer(IN:=FALSE);
                    
END_ACTION

ACTION ResetRunning_active:
                      AutomaticExecuteCompleted:=TRUE;
                    
END_ACTION

ACTION WP_Is_Metallic_active:
                      
                    
END_ACTION

ACTION TurnConveyorOff_exit:
                      Conveyor_IsSorting:=FALSE;
                    
END_ACTION

ACTION TurnConveyorOn_1_entry:
                      Timer(IN:=FALSE);
                    
END_ACTION

ACTION WP_At_Beginning_active_0:
                      Conveyor_IsSorting:=TRUE;
Conveyor_WPSorted:=FALSE;
Timer(IN:=TRUE, PT:=T#50ms);
                    
END_ACTION

ACTION LargeSortingConveyor_ACT_AutomaticExecute_Init_entry:
                      AutomaticExecuteCompleted:=FALSE;
                    
END_ACTION

ACTION Transporting_To_End_entry:
                      Timer(IN:=FALSE);
                    
END_ACTION

ACTION Conveyor_Stopping_active:
                      Conveyor_IsSorting:=FALSE;
Conveyor_WPSorted:=FALSE;
Conveyor_WPTypeChecked:=FALSE;
Conveyor_TargetChanged:=FALSE;
Conveyor_WPType_White:=FALSE;
Conveyor_WPType_Black:=FALSE;
Conveyor_WPType_Metallic:=FALSE;
Conveyor_CurrentTarget_Ramp1:=FALSE;
Conveyor_CurrentTarget_Ramp2:=FALSE;
Conveyor_CurrentTarget_Ramp3:=FALSE;

Motor.ACT_Stop();
                    
END_ACTION

ACTION Checking_WP_Type_active:
                      ACT_CheckWPType();
                    
END_ACTION

ACTION Set_Checking_False_entry:
                      Timer(IN:=FALSE);
                    
END_ACTION

ACTION Transporting_To_Ramp1_active:
                      Timer(IN:=TRUE, PT:=T#0ms);
                    
END_ACTION

ACTION Set_CahngeTarget_True_active:
                      //IF(Conveyor_CurrentTarget_Conveyor) THEN 
//Conveyor_TargetChanged:=TRUE;
//END_IF
Conveyor_TargetChanged:=TRUE;
                    
END_ACTION

ACTION Conveyor_ACT_Init_entry:
                      
                    
END_ACTION

ACTION Ramp22_active:
                      
                    
END_ACTION

ACTION Transporting_To_Ramp2_active:
                      Timer(IN:=TRUE, PT:=T#600ms);
                    
END_ACTION

ACTION TurnConveyorOf_exit:
                      
                    
END_ACTION

ACTION Wait_a_little_bit_active:
                      Timer(IN:=TRUE, PT:=T#100ms);
                    
END_ACTION

ACTION Set_ChangeTarget_FALSE_active:
                      Conveyor_CurrentTarget_Ramp1:=FALSE;
Conveyor_CurrentTarget_Ramp2:=FALSE;
Conveyor_CurrentTarget_Ramp3:=FALSE;
                    
END_ACTION

ACTION InitCompleted_FALSE_active:
                      InitCompleted:=FALSE;
                    
END_ACTION

ACTION InitCompleted_TRUE_active:
                      InitCompleted:=TRUE;
                    
END_ACTION

ACTION Changing_Target_active:
                      ACT_ChangeTarget();
                    
END_ACTION

ACTION Transporting_To_End_active:
                      Timer(IN:=TRUE, PT:=T#4000ms);
                    
END_ACTION

ACTION Sort_WP_active:
                      ACT_SortWP();
                    
END_ACTION

ACTION TurnConveyorOff_active:
                      Motor.ACT_Stop();
                    
END_ACTION

ACTION Set_Checking_False_active:
                      Timer(IN:=TRUE, PT:=T#900ms);
                    
END_ACTION

ACTION Changing_Target_entry:
                      Conveyor_TargetChanged:=FALSE;	// Franzi 2.6
                    
END_ACTION

ACTION Wait_a_little_bit_entry:
                      Timer(IN:=FALSE);
                    
END_ACTION

ACTION Checking_WP_Type_entry:
                      Conveyor_WPTypeChecked:=FALSE;
                    
END_ACTION

ACTION Sort_WP_entry:
                      Conveyor_IsSorting:=TRUE;
Conveyor_WPSorted:=FALSE;
                    
END_ACTION

ACTION Conveyor_SFCReset_active:
                      EmergencyHandeled:=TRUE;	
                    
END_ACTION

ACTION Short_Delay_entry:
                      Timer(IN:=FALSE);
                    
END_ACTION

ACTION Pusher2_Retracting_active:
                      Seperator2.ACT_Retract();
                    
END_ACTION

ACTION WP_At_Beginning_entry_0:
                      Timer(IN:=FALSE);
                    
END_ACTION

ACTION ACT_AutomaticExecute:
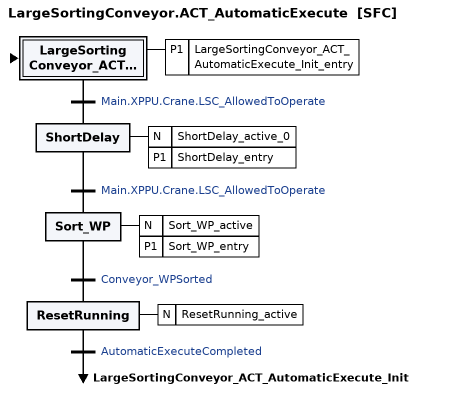
INITIAL_STEP LargeSortingConveyor_ACT_AutomaticExecute_Init:
  LargeSortingConveyor_ACT_AutomaticExecute_Init_entry(P1);
END_STEP
TRANSITION FROM LargeSortingConveyor_ACT_AutomaticExecute_Init TO ShortDelay
  := Main.XPPU.Crane.LSC_AllowedToOperate;
END_TRANSITION
STEP ShortDelay:
  ShortDelay_active_0(N);
  ShortDelay_entry(P1);
END_STEP
TRANSITION FROM ShortDelay TO Sort_WP
  := Main.XPPU.Crane.LSC_AllowedToOperate;
END_TRANSITION
STEP Sort_WP:
  Sort_WP_active(N);
  Sort_WP_entry(P1);
END_STEP
TRANSITION FROM Sort_WP TO ResetRunning
  := Conveyor_WPSorted;
END_TRANSITION
STEP ResetRunning:
  ResetRunning_active(N);
END_STEP
TRANSITION FROM ResetRunning TO LargeSortingConveyor_ACT_AutomaticExecute_Init
  := AutomaticExecuteCompleted;
END_TRANSITION
END_ACTION

ACTION ACT_EmergencyStop:
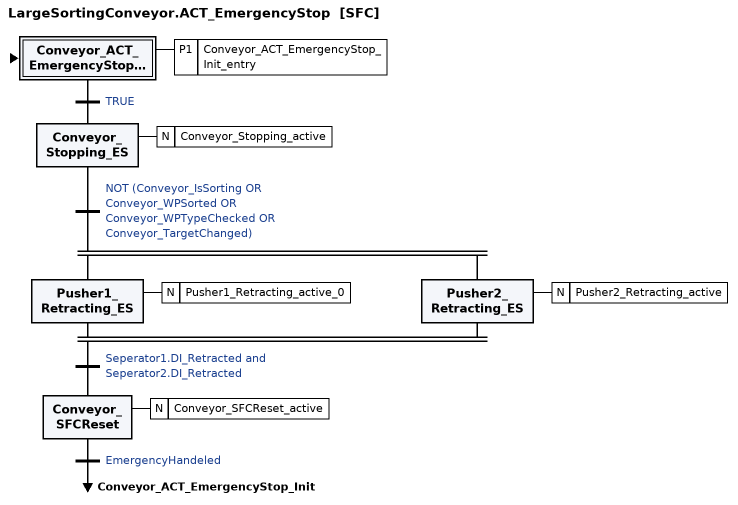
INITIAL_STEP Conveyor_ACT_EmergencyStop_Init:
  Conveyor_ACT_EmergencyStop_Init_entry(P1);
END_STEP
TRANSITION FROM Conveyor_ACT_EmergencyStop_Init TO Conveyor_Stopping_ES
  := TRUE;
END_TRANSITION
STEP Conveyor_Stopping_ES:
  Conveyor_Stopping_active(N);
END_STEP
TRANSITION FROM Conveyor_Stopping_ES TO (Pusher1_Retracting_ES, Pusher2_Retracting_ES)
  := NOT (Conveyor_IsSorting OR Conveyor_WPSorted OR Conveyor_WPTypeChecked OR Conveyor_TargetChanged);
END_TRANSITION
STEP Pusher1_Retracting_ES:
  Pusher1_Retracting_active_0(N);
END_STEP
TRANSITION FROM (Pusher1_Retracting_ES, Pusher2_Retracting_ES) TO Conveyor_SFCReset
  := Seperator1.DI_Retracted and Seperator2.DI_Retracted;
END_TRANSITION
STEP Pusher2_Retracting_ES:
  Pusher2_Retracting_active(N);
END_STEP
STEP Conveyor_SFCReset:
  Conveyor_SFCReset_active(N);
END_STEP
TRANSITION FROM Conveyor_SFCReset TO Conveyor_ACT_EmergencyStop_Init
  := EmergencyHandeled;
END_TRANSITION
END_ACTION

ACTION ACT_Init:
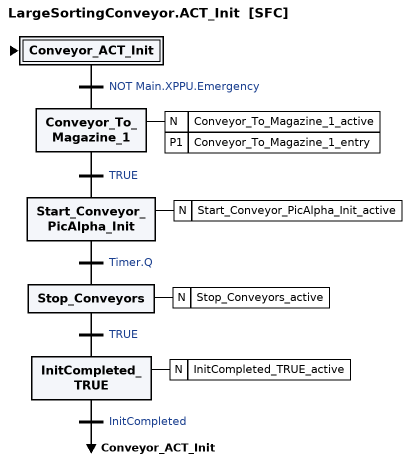
INITIAL_STEP Conveyor_ACT_Init:
END_STEP
TRANSITION FROM Conveyor_ACT_Init TO Conveyor_To_Magazine_1
  := NOT Main.XPPU.Emergency;
END_TRANSITION
STEP Conveyor_To_Magazine_1:
  Conveyor_To_Magazine_1_active(N);
  Conveyor_To_Magazine_1_entry(P1);
END_STEP
TRANSITION FROM Conveyor_To_Magazine_1 TO Start_Conveyor_PicAlpha_Init
  := TRUE;
END_TRANSITION
STEP Start_Conveyor_PicAlpha_Init:
  Start_Conveyor_PicAlpha_Init_active(N);
END_STEP
TRANSITION FROM Start_Conveyor_PicAlpha_Init TO Stop_Conveyors
  := Timer.Q;
END_TRANSITION
STEP Stop_Conveyors:
  Stop_Conveyors_active(N);
END_STEP
TRANSITION FROM Stop_Conveyors TO InitCompleted_TRUE
  := TRUE;
END_TRANSITION
STEP InitCompleted_TRUE:
  InitCompleted_TRUE_active(N);
END_STEP
TRANSITION FROM InitCompleted_TRUE TO Conveyor_ACT_Init
  := InitCompleted;
END_TRANSITION
END_ACTION

ACTION ACT_CheckWPType:
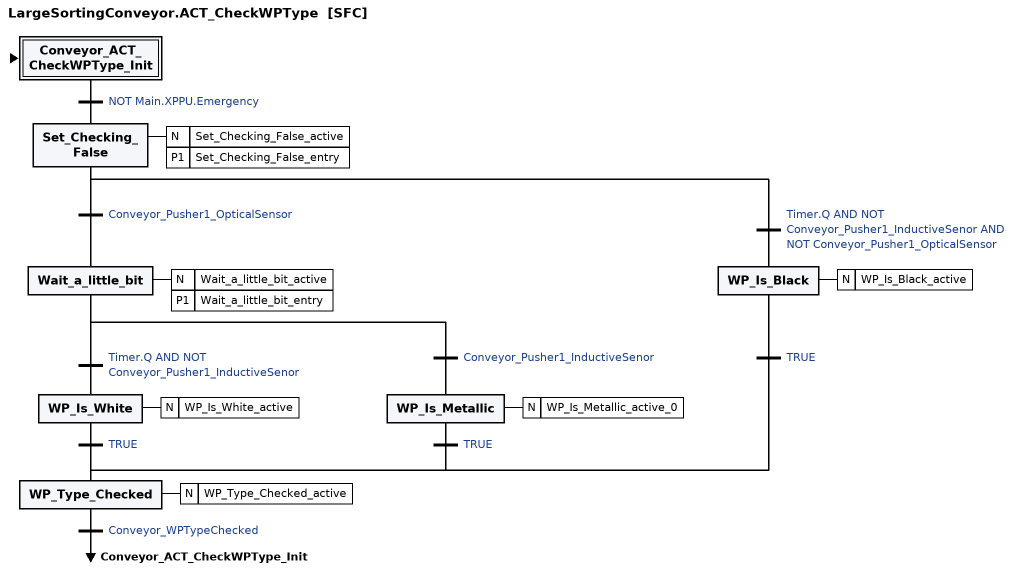
INITIAL_STEP Conveyor_ACT_CheckWPType_Init:
END_STEP
TRANSITION FROM Conveyor_ACT_CheckWPType_Init TO Set_Checking_False
  := NOT Main.XPPU.Emergency;
END_TRANSITION
STEP Set_Checking_False:
  Set_Checking_False_active(N);
  Set_Checking_False_entry(P1);
END_STEP
TRANSITION FROM Set_Checking_False TO Wait_a_little_bit
  := Conveyor_Pusher1_OpticalSensor;
END_TRANSITION
TRANSITION FROM Set_Checking_False TO WP_Is_Black
  := Timer.Q AND NOT Conveyor_Pusher1_InductiveSenor AND NOT Conveyor_Pusher1_OpticalSensor;
END_TRANSITION
STEP Wait_a_little_bit:
  Wait_a_little_bit_active(N);
  Wait_a_little_bit_entry(P1);
END_STEP
TRANSITION FROM Wait_a_little_bit TO WP_Is_White
  := Timer.Q AND NOT Conveyor_Pusher1_InductiveSenor;
END_TRANSITION
TRANSITION FROM Wait_a_little_bit TO WP_Is_Metallic
  := Conveyor_Pusher1_InductiveSenor;
END_TRANSITION
STEP WP_Is_White:
  WP_Is_White_active(N);
END_STEP
TRANSITION FROM WP_Is_White TO WP_Type_Checked
  := TRUE;
END_TRANSITION
STEP WP_Is_Metallic:
  WP_Is_Metallic_active_0(N);
END_STEP
TRANSITION FROM WP_Is_Metallic TO WP_Type_Checked
  := TRUE;
END_TRANSITION
STEP WP_Is_Black:
  WP_Is_Black_active(N);
END_STEP
TRANSITION FROM WP_Is_Black TO WP_Type_Checked
  := TRUE;
END_TRANSITION
STEP WP_Type_Checked:
  WP_Type_Checked_active(N);
END_STEP
TRANSITION FROM WP_Type_Checked TO Conveyor_ACT_CheckWPType_Init
  := Conveyor_WPTypeChecked;
END_TRANSITION
END_ACTION

ACTION ACT_SortWP:
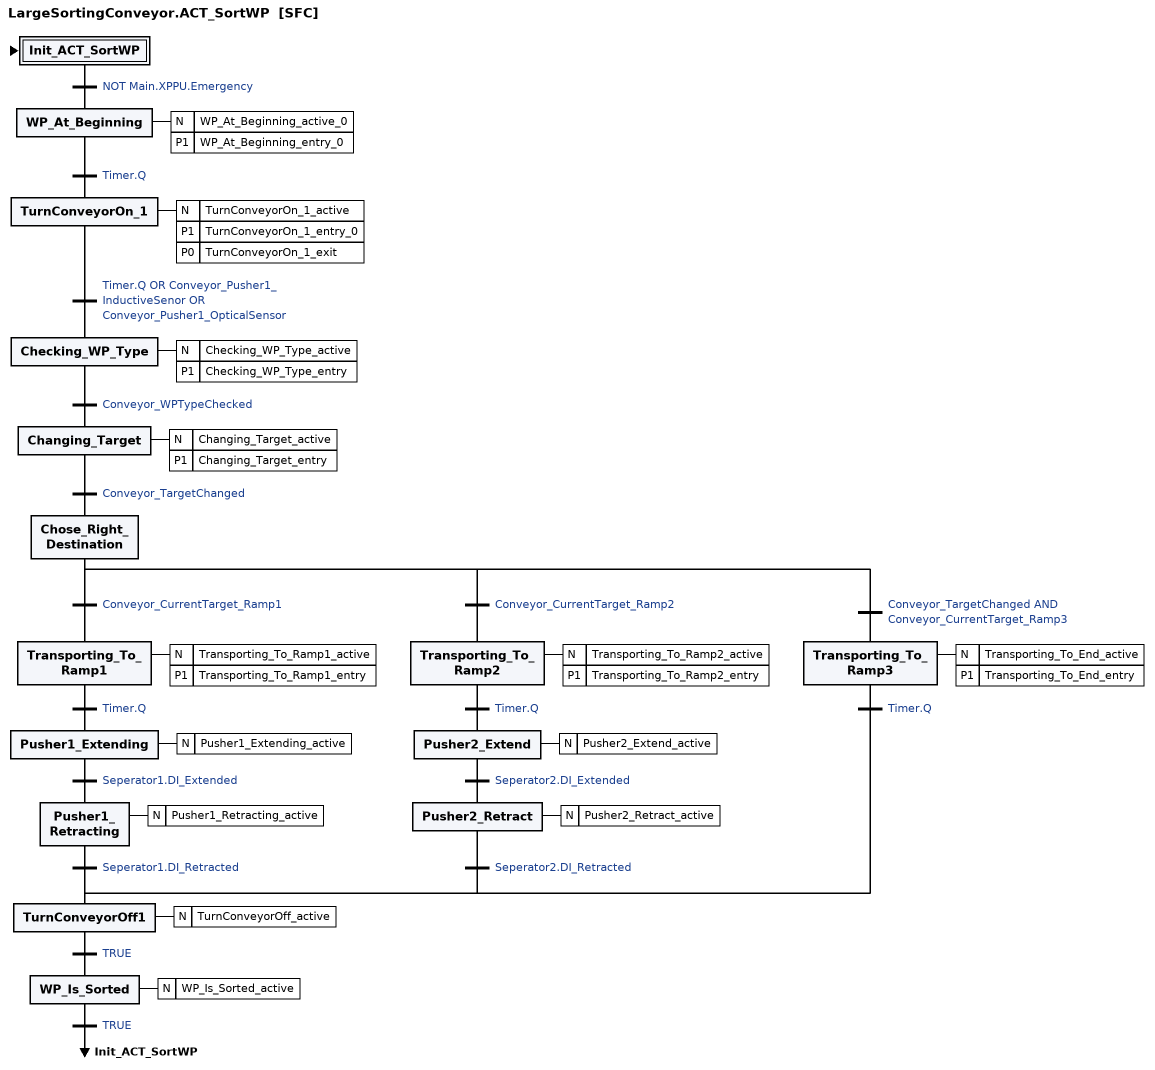
INITIAL_STEP Init_ACT_SortWP:
END_STEP
TRANSITION FROM Init_ACT_SortWP TO WP_At_Beginning
  := NOT Main.XPPU.Emergency;
END_TRANSITION
STEP WP_At_Beginning:
  WP_At_Beginning_active_0(N);
  WP_At_Beginning_entry_0(P1);
END_STEP
TRANSITION FROM WP_At_Beginning TO TurnConveyorOn_1
  := Timer.Q;
END_TRANSITION
STEP TurnConveyorOn_1:
  TurnConveyorOn_1_active(N);
  TurnConveyorOn_1_entry_0(P1);
  TurnConveyorOn_1_exit(P0);
END_STEP
TRANSITION FROM TurnConveyorOn_1 TO Checking_WP_Type
  := Timer.Q OR Conveyor_Pusher1_InductiveSenor OR Conveyor_Pusher1_OpticalSensor;
END_TRANSITION
STEP Checking_WP_Type:
  Checking_WP_Type_active(N);
  Checking_WP_Type_entry(P1);
END_STEP
TRANSITION FROM Checking_WP_Type TO Changing_Target
  := Conveyor_WPTypeChecked;
END_TRANSITION
STEP Changing_Target:
  Changing_Target_active(N);
  Changing_Target_entry(P1);
END_STEP
TRANSITION FROM Changing_Target TO Chose_Right_Destination
  := Conveyor_TargetChanged;
END_TRANSITION
STEP Chose_Right_Destination:
END_STEP
TRANSITION FROM Chose_Right_Destination TO Transporting_To_Ramp1
  := Conveyor_CurrentTarget_Ramp1;
END_TRANSITION
TRANSITION FROM Chose_Right_Destination TO Transporting_To_Ramp2
  := Conveyor_CurrentTarget_Ramp2;
END_TRANSITION
TRANSITION FROM Chose_Right_Destination TO Transporting_To_Ramp3
  := Conveyor_TargetChanged AND Conveyor_CurrentTarget_Ramp3;
END_TRANSITION
STEP Transporting_To_Ramp1:
  Transporting_To_Ramp1_active(N);
  Transporting_To_Ramp1_entry(P1);
END_STEP
TRANSITION FROM Transporting_To_Ramp1 TO Pusher1_Extending
  := Timer.Q;
END_TRANSITION
STEP Pusher1_Extending:
  Pusher1_Extending_active(N);
END_STEP
TRANSITION FROM Pusher1_Extending TO Pusher1_Retracting
  := Seperator1.DI_Extended;
END_TRANSITION
STEP Pusher1_Retracting:
  Pusher1_Retracting_active(N);
END_STEP
TRANSITION FROM Pusher1_Retracting TO TurnConveyorOff1
  := Seperator1.DI_Retracted;
END_TRANSITION
STEP Transporting_To_Ramp2:
  Transporting_To_Ramp2_active(N);
  Transporting_To_Ramp2_entry(P1);
END_STEP
TRANSITION FROM Transporting_To_Ramp2 TO Pusher2_Extend
  := Timer.Q;
END_TRANSITION
STEP Pusher2_Extend:
  Pusher2_Extend_active(N);
END_STEP
TRANSITION FROM Pusher2_Extend TO Pusher2_Retract
  := Seperator2.DI_Extended;
END_TRANSITION
STEP Pusher2_Retract:
  Pusher2_Retract_active(N);
END_STEP
TRANSITION FROM Pusher2_Retract TO TurnConveyorOff1
  := Seperator2.DI_Retracted;
END_TRANSITION
STEP Transporting_To_Ramp3:
  Transporting_To_End_active(N);
  Transporting_To_End_entry(P1);
END_STEP
TRANSITION FROM Transporting_To_Ramp3 TO TurnConveyorOff1
  := Timer.Q;
END_TRANSITION
STEP TurnConveyorOff1:
  TurnConveyorOff_active(N);
END_STEP
TRANSITION FROM TurnConveyorOff1 TO WP_Is_Sorted
  := TRUE;
END_TRANSITION
STEP WP_Is_Sorted:
  WP_Is_Sorted_active(N);
END_STEP
TRANSITION FROM WP_Is_Sorted TO Init_ACT_SortWP
  := TRUE;
END_TRANSITION
END_ACTION

ACTION ACT_GreenLampOff:
                      ConveyorGreenLamp:=FALSE;
                    
END_ACTION

ACTION ACT_GreenLampOn:
                      ConveyorGreenLamp:=TRUE;
                    
END_ACTION

ACTION ACT_WhiteLampOff:
                      ConveyorWhiteLamp:=FALSE;
                    
END_ACTION

ACTION ACT_ChangeTarget:
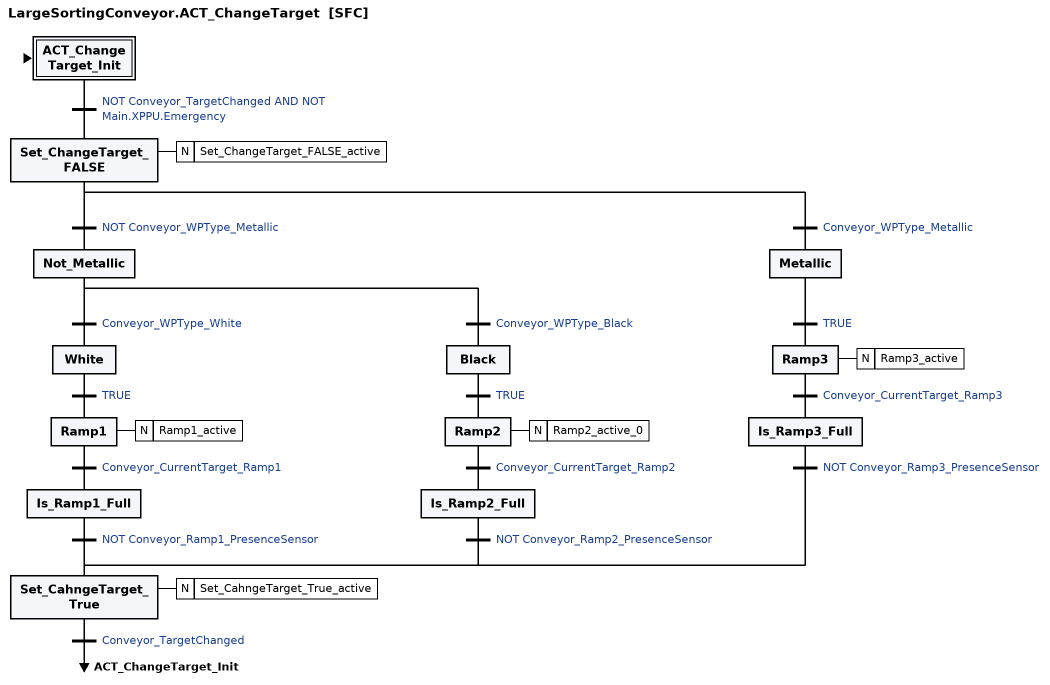
INITIAL_STEP ACT_ChangeTarget_Init:
END_STEP
TRANSITION FROM ACT_ChangeTarget_Init TO Set_ChangeTarget_FALSE
  := NOT Conveyor_TargetChanged AND NOT Main.XPPU.Emergency;
END_TRANSITION
STEP Set_ChangeTarget_FALSE:
  Set_ChangeTarget_FALSE_active(N);
END_STEP
TRANSITION FROM Set_ChangeTarget_FALSE TO Not_Metallic
  := NOT Conveyor_WPType_Metallic;
END_TRANSITION
TRANSITION FROM Set_ChangeTarget_FALSE TO Metallic
  := Conveyor_WPType_Metallic;
END_TRANSITION
STEP Not_Metallic:
END_STEP
TRANSITION FROM Not_Metallic TO White
  := Conveyor_WPType_White;
END_TRANSITION
TRANSITION FROM Not_Metallic TO Black
  := Conveyor_WPType_Black;
END_TRANSITION
STEP White:
END_STEP
TRANSITION FROM White TO Ramp1
  := TRUE;
END_TRANSITION
STEP Ramp1:
  Ramp1_active(N);
END_STEP
TRANSITION FROM Ramp1 TO Is_Ramp1_Full
  := Conveyor_CurrentTarget_Ramp1;
END_TRANSITION
STEP Is_Ramp1_Full:
END_STEP
TRANSITION FROM Is_Ramp1_Full TO Set_CahngeTarget_True
  := NOT Conveyor_Ramp1_PresenceSensor;
END_TRANSITION
STEP Black:
END_STEP
TRANSITION FROM Black TO Ramp2
  := TRUE;
END_TRANSITION
STEP Ramp2:
  Ramp2_active_0(N);
END_STEP
TRANSITION FROM Ramp2 TO Is_Ramp2_Full
  := Conveyor_CurrentTarget_Ramp2;
END_TRANSITION
STEP Is_Ramp2_Full:
END_STEP
TRANSITION FROM Is_Ramp2_Full TO Set_CahngeTarget_True
  := NOT Conveyor_Ramp2_PresenceSensor;
END_TRANSITION
STEP Metallic:
END_STEP
TRANSITION FROM Metallic TO Ramp3
  := TRUE;
END_TRANSITION
STEP Ramp3:
  Ramp3_active(N);
END_STEP
TRANSITION FROM Ramp3 TO Is_Ramp3_Full
  := Conveyor_CurrentTarget_Ramp3;
END_TRANSITION
STEP Is_Ramp3_Full:
END_STEP
TRANSITION FROM Is_Ramp3_Full TO Set_CahngeTarget_True
  := NOT Conveyor_Ramp3_PresenceSensor;
END_TRANSITION
STEP Set_CahngeTarget_True:
  Set_CahngeTarget_True_active(N);
END_STEP
TRANSITION FROM Set_CahngeTarget_True TO ACT_ChangeTarget_Init
  := Conveyor_TargetChanged;
END_TRANSITION
END_ACTION

ACTION ACT_WhiteLampOn:
                      ConveyorWhiteLamp:=TRUE;

                    
END_ACTION

ACTION Ramp2_active_0:
                      Conveyor_CurrentTarget_Ramp2:=TRUE;
                    
END_ACTION

ACTION Ramp3_active:
                      Conveyor_CurrentTarget_Ramp3:=TRUE;
                    
END_ACTION
END_FUNCTION_BLOCK

FUNCTION_BLOCK Stack
VAR_INPUT	
	Seperator : MonostableCylinder;	
	//Software
	SFCReset : BOOL;
	InitCompleted : BOOL;
	EmergencyHandeled : BOOL;	
END_VAR
VAR_OUTPUT	
	//Software
	Stack_WPType_White : BOOL;
	Stack_WPType_Black : BOOL;
	Stack_WPType_Metallic : BOOL;
	Stack_WPWeight_Light : BOOL;
	Stack_WPWeight_Medium : BOOL;
	Stack_WPWeight_Heavy : BOOL;
	Stack_WPProvided : BOOL;	
END_VAR
VAR
	//Hardware
	Stack_WorkpieceReady AT %I* : BOOL;
	Stack_InductiveSensor AT %I* : BOOL;
	Stack_OpticalSensor AT %I* : BOOL;
	Stack_WPWeight AT %I* : INT;
	Stack_StartButton AT %I* : BOOL;
	Stack_EmergencyStop AT %I* : BOOL;	
	StackGreenLamp AT %Q* : BOOL;
	StackWhiteLamp AT %Q* : BOOL;
	
	//Software
	Timer : TON;		
END_VAR

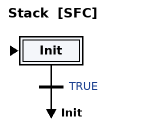
INITIAL_STEP Init:
END_STEP
TRANSITION FROM Init TO Init
  := TRUE;
END_TRANSITION

ACTION ACT_GreenLampOn:
                      StackGreenLamp:=TRUE;
                    
END_ACTION

ACTION ACT_GreenLampOff:
                      StackGreenLamp:=FALSE;
                    
END_ACTION

ACTION ACT_WhiteLampOff:
                      StackWhiteLamp:=FALSE;
                    
END_ACTION

ACTION ACT_WhiteLampOn:
                      StackWhiteLamp:=TRUE;
StackGreenLamp:=FALSE;
                    
END_ACTION

ACTION ACT_ProvideWP:
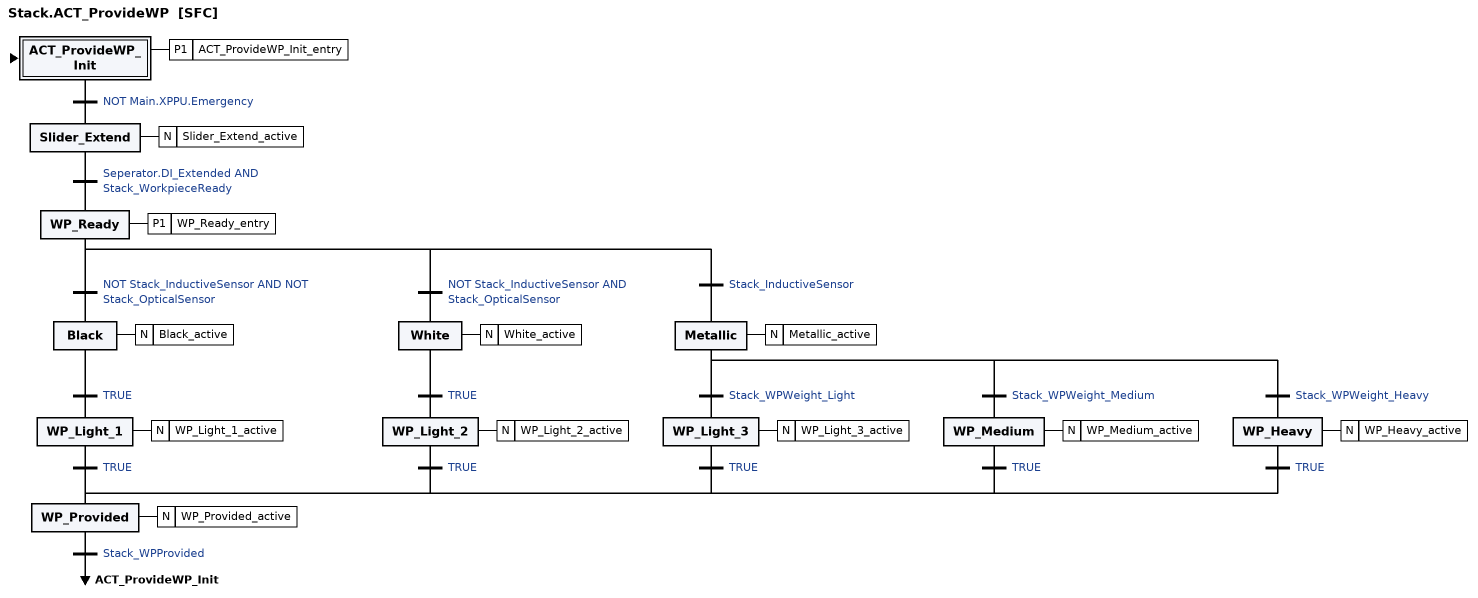
INITIAL_STEP ACT_ProvideWP_Init:
  ACT_ProvideWP_Init_entry(P1);
END_STEP
TRANSITION FROM ACT_ProvideWP_Init TO Slider_Extend
  := NOT Main.XPPU.Emergency;
END_TRANSITION
STEP Slider_Extend:
  Slider_Extend_active(N);
END_STEP
TRANSITION FROM Slider_Extend TO WP_Ready
  := Seperator.DI_Extended AND Stack_WorkpieceReady;
END_TRANSITION
STEP WP_Ready:
  WP_Ready_entry(P1);
END_STEP
TRANSITION FROM WP_Ready TO Black
  := NOT Stack_InductiveSensor AND NOT Stack_OpticalSensor;
END_TRANSITION
TRANSITION FROM WP_Ready TO White
  := NOT Stack_InductiveSensor AND Stack_OpticalSensor;
END_TRANSITION
TRANSITION FROM WP_Ready TO Metallic
  := Stack_InductiveSensor;
END_TRANSITION
STEP Black:
  Black_active(N);
END_STEP
TRANSITION FROM Black TO WP_Light_1
  := TRUE;
END_TRANSITION
STEP WP_Light_1:
  WP_Light_1_active(N);
END_STEP
TRANSITION FROM WP_Light_1 TO WP_Provided
  := TRUE;
END_TRANSITION
STEP White:
  White_active(N);
END_STEP
TRANSITION FROM White TO WP_Light_2
  := TRUE;
END_TRANSITION
STEP WP_Light_2:
  WP_Light_2_active(N);
END_STEP
TRANSITION FROM WP_Light_2 TO WP_Provided
  := TRUE;
END_TRANSITION
STEP Metallic:
  Metallic_active(N);
END_STEP
TRANSITION FROM Metallic TO WP_Light_3
  := Stack_WPWeight_Light;
END_TRANSITION
TRANSITION FROM Metallic TO WP_Medium
  := Stack_WPWeight_Medium;
END_TRANSITION
TRANSITION FROM Metallic TO WP_Heavy
  := Stack_WPWeight_Heavy;
END_TRANSITION
STEP WP_Light_3:
  WP_Light_3_active(N);
END_STEP
TRANSITION FROM WP_Light_3 TO WP_Provided
  := TRUE;
END_TRANSITION
STEP WP_Medium:
  WP_Medium_active(N);
END_STEP
TRANSITION FROM WP_Medium TO WP_Provided
  := TRUE;
END_TRANSITION
STEP WP_Heavy:
  WP_Heavy_active(N);
END_STEP
TRANSITION FROM WP_Heavy TO WP_Provided
  := TRUE;
END_TRANSITION
STEP WP_Provided:
  WP_Provided_active(N);
END_STEP
TRANSITION FROM WP_Provided TO ACT_ProvideWP_Init
  := Stack_WPProvided;
END_TRANSITION
END_ACTION

ACTION Slider_Extend_active:
                      Seperator.ACT_Extend();
                    
END_ACTION

ACTION Crane_To_Magazine_active:
                      Main.XPPU.Crane.ACT_MoveToStack();
                    
END_ACTION

ACTION Provide_WP_active:
                      ACT_ProvideWP();
                    
END_ACTION

ACTION WP_Ready_entry:
                      Stack_WPType_White:=FALSE;
Stack_WPType_Black:=FALSE;
Stack_WPType_Metallic:=FALSE;
Stack_WPWeight_Light:=FALSE;
Stack_WPWeight_Medium:=FALSE;
Stack_WPWeight_Heavy:=FALSE;
                    
END_ACTION

ACTION Stack_Retracing_active:
                      Seperator.ACT_Retract();
                    
END_ACTION

ACTION Short_Delay_active:
                      Timer(IN:=TRUE, PT:=T#50ms);
                    
END_ACTION

ACTION Slider_Move_In_active:
                      Seperator.ACT_Retract();
                    
END_ACTION

ACTION Short_Delay_entry:
                      Timer(IN:=FALSE);
                    
END_ACTION

ACTION WP_Heavy_active:
                      Stack_WPWeight_Heavy:=TRUE;
                    
END_ACTION

ACTION WP_Light_2_active:
                      Stack_WPWeight_Light:=TRUE;
                    
END_ACTION

ACTION Set_WP_Parameters_active:
                      IF(NOT Stack_InductiveSensor AND NOT Stack_OpticalSensor)THEN
	Stack_WPType_Black:=TRUE;
	Stack_WPType_White:=FALSE;
	Stack_WPType_Metallic:=FALSE;
ELSIF(NOT Stack_InductiveSensor AND Stack_OpticalSensor)THEN
	Stack_WPType_Black:=FALSE;
	Stack_WPType_White:=TRUE;
	Stack_WPType_Metallic:=FALSE;
ELSIF(Stack_InductiveSensor)THEN
	Stack_WPType_Black:=FALSE;
	Stack_WPType_White:=FALSE;
	Stack_WPType_Metallic:=TRUE;
END_IF

IF(Stack_WPType_Black OR Stack_WPType_White OR(Stack_WPType_Metallic AND Stack_WPWeight < 12000))THEN
	Stack_WPWeight_Light:=TRUE;
	Stack_WPWeight_Medium:=FALSE;
	Stack_WPWeight_Heavy:=FALSE;
ELSIF(12000<Stack_WPWeight AND Stack_WPWeight<=24000)THEN
	Stack_WPWeight_Light:=FALSE;
	Stack_WPWeight_Medium:=TRUE;
	Stack_WPWeight_Heavy:=FALSE;	
ELSIF(24000<=Stack_WPWeight)THEN
	Stack_WPWeight_Light:=FALSE;
	Stack_WPWeight_Medium:=FALSE;
	Stack_WPWeight_Heavy:=TRUE;	
END_IF

Stack_WPProvided:=TRUE;
                    
END_ACTION

ACTION Metallic_active:
                      Stack_WPType_Metallic:=TRUE;
IF(Stack_WPWeight < 12000)THEN
	Stack_WPWeight_Light:=TRUE;
END_IF
IF(12000<Stack_WPWeight AND Stack_WPWeight<=24000)THEN
	Stack_WPWeight_Medium:=TRUE;
END_IF
IF(24000<=Stack_WPWeight)THEN
	Stack_WPWeight_Heavy:=TRUE;
END_IF

                    
END_ACTION

ACTION WP_Allreday_Provided_active:
                      
                    
END_ACTION

ACTION PutDown_WP_active:
                      Main.XPPU.Crane.ACT_PutDownWP();
                    
END_ACTION

ACTION Stack_SFCReset_active:
                       EmergencyHandeled:=TRUE;		
                    
END_ACTION

ACTION Magazine_ACT_EmergencyStop_Init_entry:
                      StackGreenLamp:=FALSE;
StackWhiteLamp:=FALSE;
                    
END_ACTION

ACTION WP_Provided_active:
                      Stack_WPProvided:=TRUE;
                    
END_ACTION

ACTION WP_Light_1_active:
                      Stack_WPWeight_Light:=TRUE;
                    
END_ACTION

ACTION Black_active:
                      Stack_WPType_Black:=TRUE;
                    
END_ACTION

ACTION InitCompleted_TRUE_active:
                      InitCompleted:=TRUE;
                    
END_ACTION

ACTION Stack_ACT_Init_entry:
                      

                    
END_ACTION

ACTION WP_Light_3_active:
                      Stack_WPWeight_Light:=TRUE;
                    
END_ACTION

ACTION WP_Medium_active:
                      Stack_WPWeight_Medium:=TRUE;
                    
END_ACTION

ACTION Slider_Move_In_2_active:
                      Seperator.ACT_Retract();
                    
END_ACTION

ACTION WP_To_Conveyor_active:
                      Main.XPPU.Crane.ACT_MoveToConveyor();
                    
END_ACTION

ACTION Stack_Retracting_active:
                      Stack_WPType_White:=FALSE;
Stack_WPType_Black:=FALSE;
Stack_WPType_Metallic:=FALSE;
Stack_WPWeight_Light:=FALSE;
Stack_WPWeight_Medium:=FALSE;
Stack_WPWeight_Heavy:=FALSE;
Stack_WPProvided:=FALSE;

Seperator.ACT_Retract();
                    
END_ACTION

ACTION SortWP_Init_active:
                      Main.XPPU.LargeSortingConveyor.ACT_SortWP();
                    
END_ACTION

ACTION Pick_Up_WP_active:
                      Main.XPPU.Crane.ACT_PickUpWP();
                    
END_ACTION

ACTION White_active:
                      Stack_WPType_White:=TRUE;
                    
END_ACTION

ACTION Retract_Cylinder_Init_active:
                      Seperator.ACT_Retract();
                    
END_ACTION

ACTION ACT_ProvideWP_Init_entry:
                      Stack_WPProvided:=FALSE;
                    
END_ACTION

ACTION ACT_EmergencyStop:
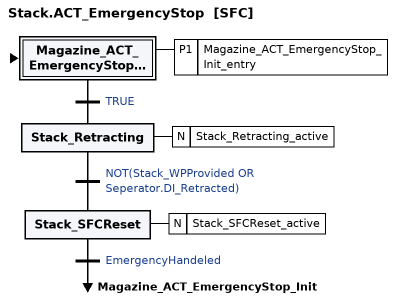
INITIAL_STEP Magazine_ACT_EmergencyStop_Init:
  Magazine_ACT_EmergencyStop_Init_entry(P1);
END_STEP
TRANSITION FROM Magazine_ACT_EmergencyStop_Init TO Stack_Retracting
  := TRUE;
END_TRANSITION
STEP Stack_Retracting:
  Stack_Retracting_active(N);
END_STEP
TRANSITION FROM Stack_Retracting TO Stack_SFCReset
  := NOT(Stack_WPProvided OR Seperator.DI_Retracted);
END_TRANSITION
STEP Stack_SFCReset:
  Stack_SFCReset_active(N);
END_STEP
TRANSITION FROM Stack_SFCReset TO Magazine_ACT_EmergencyStop_Init
  := EmergencyHandeled;
END_TRANSITION
END_ACTION

ACTION ACT_AutomaticExecute:
